{attribute addProperty BoxType "ATH2000-5250-0022"}
{attribute addProperty Id "BinaryDataAT %I*ARRAY [0..63] OF BYTE00"}
{attribute addProperty CRC "461638819"}
{attribute addProperty SizeInBites "0"}
{attribute addProperty SizeInBytes "0"}
TYPE FB_Inputs_1B840CA3 :
STRUCT
	{attribute addProperty Name "BinaryData"}
	BinaryData AT %I* : ARRAY [0..63] OF BYTE;
END_STRUCT
END_TYPE

(* stored: Version 1.2.0.0, ProductVersion 3.1.4024.9
   DUT FB_Inputs_1B840CA3: Id {898d2637-3024-461f-ba39-8f28ab27ada3} *)
